Yaskawa INFORM job: CLEAN-R1.JBI

/JOB
//NAME CLEAN-R1
///FOLDERNAME CLEAN
//POS
///NPOS 22,22,0,0,0,0
///TOOL 0
///POSTYPE PULSE
///PULSE
C00000=-39727,-76224,-106676,19950,71810,76872
C00001=2508,0,0,0,0,4169
C00002=32571,-80067,-84751,-11816,58952,90735
C00003=41115,93452,-30342,-19926,115521,85678
C00004=28599,109925,-13759,-12658,112881,84157
C00005=28301,105457,-14309,-12299,110948,84323
C00006=28966,99224,-20084,-13542,107459,84155
C00007=29027,99166,-20392,-13590,107618,84144
C00008=28599,108424,-14443,-12622,112541,84195
C00009=34011,109773,-12073,-16636,107751,84808
C00010=32816,112629,-5671,-14598,109695,85231
C00011=32618,110353,-5730,-14378,108579,85337
C00012=32545,109523,-5728,-14298,108158,85375
C00013=32618,110353,-5730,-14378,108579,85337
C00014=32816,112629,-5671,-14598,109695,85231
C00015=34011,109773,-12073,-16636,107751,84808
C00016=38810,111241,-7992,-19438,105697,85727
C00017=36913,114349,813,-16982,106196,86149
C00018=37169,116704,797,-17245,107389,86018
C00019=39968,92120,-23778,-21749,94252,85800
C00020=46315,71110,-54300,-23622,119041,85704
C00021=32571,-80067,-84751,-11816,58952,90735
BC00000=295327,674570,1075173
BC00001=0,0,0
BC00002=204899,578,820586
BC00003=204899,578,1075157
BC00004=204899,578,1075157
BC00005=204899,578,1075157
BC00006=204899,578,1075157
BC00007=204899,578,1075157
BC00008=204899,578,1075157
BC00009=204899,578,1075157
BC00010=204899,578,1075157
BC00011=204899,578,1075157
BC00012=204899,578,1075157
BC00013=204899,578,1075157
BC00014=204899,578,1075157
BC00015=204899,578,1075157
BC00016=204899,578,1075157
BC00017=204894,578,1075156
BC00018=204894,578,1075156
BC00019=204894,578,1075156
BC00020=204899,578,1075157
BC00021=204899,578,820586
//INST
///DATE 2024/02/03 14:51
///ATTR SC,RW
///GROUP1 RB1,BS1
///LVARS 0,5,0,0,0,3,3,0
NOP
MOVJ C00000 BC00000 VJ=10.00
SFTOF
'********************************
'Please check position before
'running in play-mode
'********************************
'#Output - Cleaning Motor
SET LI000 14
'#Output - Cleaning Oil
SET LI001 15
'#Output - Wirecut
SET LI002 16
'#Output - Wirefeeder Forward
SET LI003 4095
'#Output - Torch Blow out
SET LI004 4091
'********************************
REFP 1 C00001 BC00001
GETS LPX001 $PX011
CNVRT LPX001 LPX001 RF
GETS LPX002 $PX001
CNVRT LPX002 LPX002 RF
SUB LBP002 LBP001
'Comment out axis to shift
SETE LBP002 (1) 0
COMM SETE LBP002 (2) 0
SETE LBP002 (3) 0
SFTON LBP002
'********************************
'SAFE POS
PAUSE IF IN#(1563)=OFF
MOVJ C00002 BC00002 VJ=50.00
MOVJ C00003 BC00003 VJ=50.00
'WIRECUT
MOVJ C00004 BC00004 VJ=50.00
'WIREFEED OUTPUT
PULSE OT#(LI003) T=0.80
MOVL C00005 BC00005 V=75.0
MOVL C00006 BC00006 V=20.0
TIMER T=0.20
DOUT OT#(LI002) ON
TIMER T=1.00
MOVL C00007 BC00007 V=20.0
MOVL C00008 BC00008 V=75.0
DOUT OT#(LI002) OFF
'CLEANING MOTOR
MOVJ C00009 BC00009 VJ=50.00
MOVL C00010 BC00010 V=75.0
'CLEANING AIR
DOUT OT#(LI004) ON
MOVL C00011 BC00011 V=20.0
TIMER T=0.20
DOUT OT#(LI000) ON
TIMER T=0.50
MOVL C00012 BC00012 V=20.0
TIMER T=0.50
MOVL C00013 BC00013 V=20.0
TIMER T=0.20
DOUT OT#(LI000) OFF
TIMER T=0.50
DOUT OT#(LI004) OFF
MOVL C00014 BC00014 V=20.0
MOVL C00015 BC00015 V=75.0
'CLEANING OIL
MOVJ C00016 BC00016 VJ=50.00
MOVL C00017 BC00017 V=75.0
PULSE OT#(LI001) T=0.20
TIMER T=1.00
MOVL C00018 BC00018 V=75.0
'CLEANING AIR
PULSE OT#(LI004) T=1.00
TIMER T=1.00
MOVJ C00019 BC00019 VJ=25.00
'SAFE POS
MOVJ C00020 BC00020 VJ=25.00
MOVJ C00021 BC00021 VJ=50.00
SFTOF
'********************************
'*         CLEANING JOB         *
'*      __ __ _____ _____       *
'*     |  |  |   | | __  |      *
'*     |_   _| | | |    -|      *
'*       |_| |_|___|__|__|      *
'*        YRC Multi Base        *
'*       rev 4. 2021-10-12      *
'********************************
END
